FUNCTION_BLOCK FB_TcMessageSuccess EXTENDS FB_TcMessage
VAR
END_VAR

METHOD FB_init : BOOL
VAR_INPUT
	bInitRetains: BOOL; // if TRUE, the retain variables are initialized (warm start / cold start)
	bInCopyCode: BOOL; // if TRUE, the instance afterwards gets moved into the copy code (online change)
END_VAR
VAR
END_VAR
IF NOT bInCopyCode THEN
	SUPER^.CreateEx(Tc3_EventLogger.SUCCESS_EVENT, 0);
END_IF
END_METHOD

END_FUNCTION_BLOCK

(* stored: POU FB_TcMessageSuccess: Id 80530bba-1e56-41aa-8c40-4f363c2dfc2f, SpecialFunc None
   Method FB_init: Id 927a351d-1868-4929-a893-ae85e68e52a0 *)
